// TIA Portal project "eldar_haseljic_TIA_seminarski" (V14)

(* hardware
DEVICE "S71500/ET200MP-Station_1"  S7-1500 station
   slot 0: "Profilschiene_0"  6ES7 590-1***0-0AA0
   slot 1: "PLC_1"  CPU 1511-1 PN  6ES7 511-1AK00-0AB0  V1.8
   slot 2: "AI 8xU/I/RTD/TC ST_1"  AI 8xU/I/RTD/TC ST  6ES7 531-7KF00-0AB0  V2.0
   slot 3: "AI 8xU/I/RTD/TC ST_2"  AI 8xU/I/RTD/TC ST  6ES7 531-7KF00-0AB0  V2.0
   slot 4: "AI 8xU/I/RTD/TC ST_3"  AI 8xU/I/RTD/TC ST  6ES7 531-7KF00-0AB0  V2.0
   slot 5: "AI 8xU/I/RTD/TC ST_4"  AI 8xU/I/RTD/TC ST  6ES7 531-7KF00-0AB0  V2.0
   slot 6: "DI 16x24VDC BA_1"  DI 16x24VDC BA  6ES7 521-1BH10-0AA0  V1.0
*)

// ===== PLC "PLC_1"  CPU 1511-1 PN =====

VAR_GLOBAL   // PLC tag table "Standard-Variablentabelle"
   "Clock_Byte" AT %MB0 : Byte;
   "Clock_10Hz" AT %M0.0 : Bool;
   "Clock_5Hz" AT %M0.1 : Bool;
   "Clock_2.5Hz" AT %M0.2 : Bool;
   "Clock_2Hz" AT %M0.3 : Bool;
   "Clock_1.25Hz" AT %M0.4 : Bool;
   "Clock_1Hz" AT %M0.5 : Bool;
   "Clock_0.625Hz" AT %M0.6 : Bool;
   "Clock_0.5Hz" AT %M0.7 : Bool;
   "Start_Button_1" AT %I0.0 : Bool;
   "Stop_Button_1" AT %I0.1 : Bool;
   "Stop_Button_2" AT %I0.2 : Bool;
   "Diffuse_Senzor_1" AT %I0.3 : Bool;
   "Diffuse_Senzor_2" AT %I0.4 : Bool;
   "Diffuse_Senzor_3" AT %I0.5 : Bool;
   "Belt_Conveyor(4m)" AT %Q0.0 : Bool;
   "Belt_Conveyor(6m)" AT %Q0.1 : Bool;
   "Stack_Light_1(Red)" AT %Q0.2 : Bool;
   "Stack_Light_1(Green)" AT %Q0.3 : Bool;
   "Stack_Light_1(Yellow)" AT %Q0.4 : Bool;
   "Stack_Light_2(Red)" AT %Q0.5 : Bool;
   "Stack_Light_2(Yellow)" AT %Q0.6 : Bool;
   "Stack_Light_2(Green)" AT %Q0.7 : Bool;
END_VAR

DATA_BLOCK "Ormar_DB"   // DB2
{ S7_Optimized_Access := 'TRUE' }
VERSION : 0.1
// stored: InstanceOfName Ormar
"Ormar"
BEGIN
END_DATA_BLOCK

// folder: System blocks/Program resources

DATA_BLOCK "IEC_Counter_0_DB"   // DB1
{ S7_Optimized_Access := 'TRUE' }
AUTHOR : Simatic
FAMILY : IEC
NAME : CNTR
VERSION : 1.0
// stored: InstanceOfName IEC_COUNTER
"IEC_COUNTER"
BEGIN
END_DATA_BLOCK

DATA_BLOCK "IEC_Counter_0_DB_1"   // DB3
{ S7_Optimized_Access := 'TRUE' }
AUTHOR : Simatic
FAMILY : IEC
NAME : CNTR
VERSION : 1.0
// stored: InstanceOfName IEC_COUNTER
"IEC_COUNTER"
BEGIN
END_DATA_BLOCK

// folder: (top level)

FUNCTION_BLOCK "Ormar"   // FB1, LAD
{ S7_Optimized_Access := 'TRUE' }
VERSION : 0.1
   VAR_INPUT
      Start : Bool;
      Stop1 : Bool;
      Stop2 : Bool;
      Senzor1 : Bool;
      Senzor2 : Bool;
      Senzor3 : Bool;
   END_VAR
   VAR_OUTPUT
      Zelena1 : Bool;
      Zelena2 : Bool;
      Crvena1 : Bool;
      Crvena2 : Bool;
      Zuta1 : Bool;
      Zuta2 : Bool;
   END_VAR
   VAR_IN_OUT
      Traka1 : Bool;
      Traka2 : Bool;
   END_VAR
BEGIN

REGION Network 1
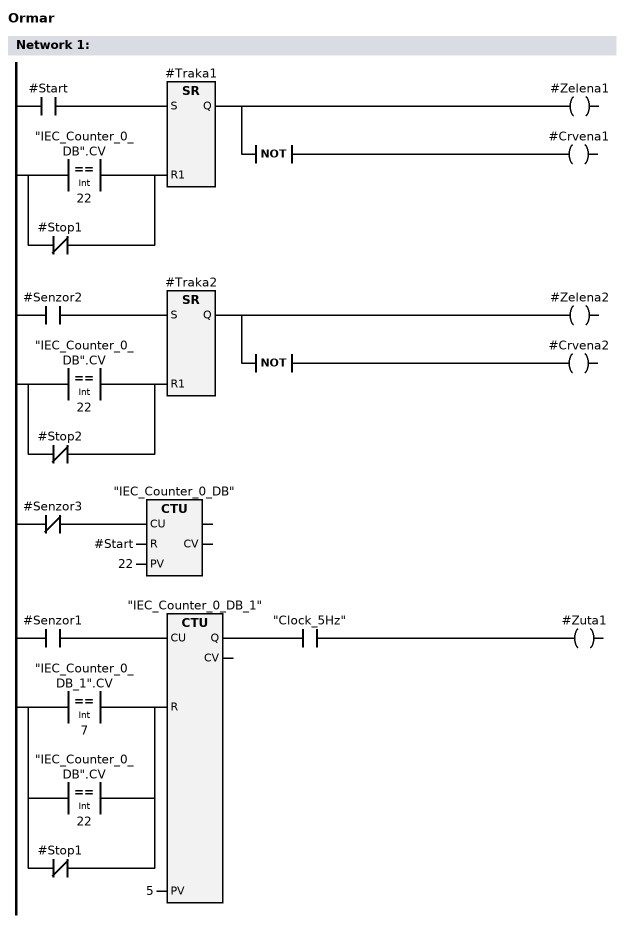
   IF #Start THEN
       #Traka1 := TRUE;   // SR flip-flop
   END_IF;
   IF ("IEC_Counter_0_DB".CV = 22) OR NOT #Stop1 THEN #Traka1 := FALSE; END_IF;
   #Zelena1 := #Traka1;
   #Crvena1 := NOT #Traka1;
   IF #Senzor2 THEN
       #Traka2 := TRUE;   // SR flip-flop
   END_IF;
   IF ("IEC_Counter_0_DB".CV = 22) OR NOT #Stop2 THEN #Traka2 := FALSE; END_IF;
   #Zelena2 := #Traka2;
   #Crvena2 := NOT #Traka2;
   "IEC_Counter_0_DB".CTU(CU := NOT #Senzor3, R := #Start, PV := 22);
   "IEC_Counter_0_DB_1".CTU(CU := #Senzor1,
                           R := ("IEC_Counter_0_DB_1".CV = 7) OR ("IEC_Counter_0_DB".CV = 22) OR NOT #Stop1,
                           PV := 5);
   #Zuta1 := "IEC_Counter_0_DB_1".Q AND "Clock_5Hz";
END_REGION
END_FUNCTION_BLOCK

FUNCTION "Inicijalizacija" : Void   // FC1, LAD
{ S7_Optimized_Access := 'TRUE' }
VERSION : 0.1
   VAR_OUTPUT
      Crvena1 : Bool;
      Crvena2 : Bool;
   END_VAR
BEGIN

REGION Network 1
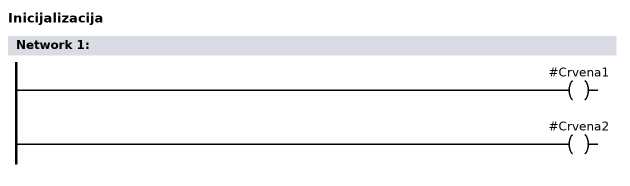
   RUNG wire#powerrail
      Coil( #Crvena1 )
   END_RUNG
   RUNG wire#powerrail
      Coil( #Crvena2 )
   END_RUNG
   // the same network as SCL:
   #Crvena1 := TRUE;
   #Crvena2 := TRUE;
END_REGION
END_FUNCTION

FUNCTION "MHJ-PLC-Lab-Function-S71500" : Void   // FC9000, SCL
{ S7_Optimized_Access := 'TRUE' }
VERSION : 0.1
   VAR_TEMP
      Value : Byte;
      ForCounter : Int;
   END_VAR
   VAR CONSTANT
      Value_01_DW : DWord := 16#1223_5486;
      Value_02_DW : DWord := 16#A6C9_D1F5;
   END_VAR
BEGIN

   #Value:=PEEK(area := 16#82,
        dbNumber := 0,
        byteOffset := 511);
   #Value := #Value + 1;

   POKE(area := 16#82,
        dbNumber := 0,
        byteOffset := 511,
        value := #Value);

   POKE(area := 16#82,
        dbNumber := 0,
        byteOffset := 1016,
        value := #Value_01_DW);
   POKE(area := 16#82,
        dbNumber := 0,
        byteOffset := 1020,
        value := #Value_02_DW);

   FOR #ForCounter := 0 TO 63 DO
       #Value:=PEEK(area := 16#1,
            dbNumber := 0,
            byteOffset := #ForCounter);
       POKE(area := 16#81,
            dbNumber := 0,
            byteOffset := #ForCounter,
            value := #Value);
   END_FOR;
   #Value := PEEK(area := 16#1,
                  dbNumber := 0,
                  byteOffset := 512);
   POKE(area := 16#82,
        dbNumber := 0,
        byteOffset := 512,
        value := #Value);
END_FUNCTION

ORGANIZATION_BLOCK "Main"   // OB1, LAD, ProgramCycle
TITLE = "Main Program Sweep (Cycle)"
{ S7_Optimized_Access := 'TRUE' }
VERSION : 0.1
   VAR_INPUT
      Initial_Call : Bool;   // Initial call of this OB
      Remanence : Bool;   // =True, if remanent data are available
   END_VAR
   VAR_TEMP   // added for the SCL form of the ladder/FBD networks
      _w1 : Bool;
   END_VAR
BEGIN

REGION Network 1
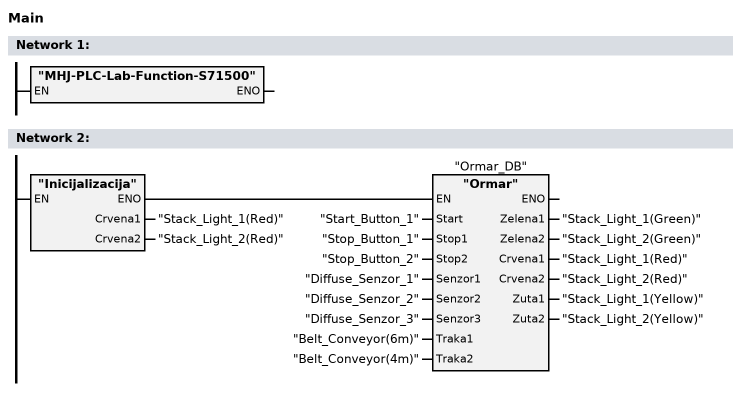
   RUNG wire#powerrail
      "MHJ-PLC-Lab-Function-S71500"()
   END_RUNG
   // the same network as SCL:
   "MHJ-PLC-Lab-Function-S71500"();
END_REGION

REGION Network 2
   RUNG wire#powerrail
      "Inicijalizacija"(Crvena1 => "Stack_Light_1(Red)", Crvena2 => "Stack_Light_2(Red)")
      "Ormar_DB"(Start := "Start_Button_1", Stop1 := "Stop_Button_1", Stop2 := "Stop_Button_2", Senzor1 := "Diffuse_Senzor_1", Senzor2 := "Diffuse_Senzor_2", Senzor3 := "Diffuse_Senzor_3", Traka1 := "Belt_Conveyor(6m)", Traka2 := "Belt_Conveyor(4m)", Zelena1 => "Stack_Light_1(Green)", Zelena2 => "Stack_Light_2(Green)", Crvena1 => "Stack_Light_1(Red)", Crvena2 => "Stack_Light_2(Red)", Zuta1 => "Stack_Light_1(Yellow)", Zuta2 => "Stack_Light_2(Yellow)")
   END_RUNG
   // the same network as SCL:
   "Inicijalizacija"(Crvena1 => "Stack_Light_1(Red)", Crvena2 => "Stack_Light_2(Red)", ENO => #_w1);
   IF #_w1 THEN
       "Ormar_DB"(Start := "Start_Button_1",   // "Ormar"
                  Stop1 := "Stop_Button_1",
                  Stop2 := "Stop_Button_2",
                  Senzor1 := "Diffuse_Senzor_1",
                  Senzor2 := "Diffuse_Senzor_2",
                  Senzor3 := "Diffuse_Senzor_3",
                  Traka1 := "Belt_Conveyor(6m)",
                  Traka2 := "Belt_Conveyor(4m)",
                  Zelena1 => "Stack_Light_1(Green)",
                  Zelena2 => "Stack_Light_2(Green)",
                  Crvena1 => "Stack_Light_1(Red)",
                  Crvena2 => "Stack_Light_2(Red)",
                  Zuta1 => "Stack_Light_1(Yellow)",
                  Zuta2 => "Stack_Light_2(Yellow)");
   END_IF;
END_REGION
END_ORGANIZATION_BLOCK